// TIA Portal V18 export
// export: Created 2025-12-01T17:50:27.3546256Z, ExportSetting None, DisplayName Totally Integrated Automation Portal, DisplayVersion V18 Update 5, DisplayName TIA Portal Openness, DisplayVersion V18 Update 5, DisplayName TIA Portal Teamcenter Gateway, DisplayVersion V18, DisplayName TIA Portal Version Control Interface, DisplayVersion V18, DisplayName STEP 7 Professional, DisplayVersion V18 Update 5, DisplayName STEP 7 Safety, DisplayVersion V18, DisplayName WinCC Professional, DisplayVersion V18 Update 5
FUNCTION "CheckData" : Void   // FC4023, SCL
{ S7_Optimized_Access := 'FALSE' }
// stored: AutoNumber false, SetENOAutomatically false
   VAR_INPUT
      DBNo : Int;
      DBBNO : Int;
      ByteLenth : Int;
   END_VAR
   VAR_OUTPUT
      AlarmON : Bool;
   END_VAR
   VAR_TEMP
      AlarmByte : Int;
      tByte : Int;
   END_VAR
BEGIN
   #AlarmON := 0;
   #AlarmByte := 0;
   IF #ByteLenth>0 THEN
       FOR #tByte:=0 TO #ByteLenth-1 DO
           IF PEEK_BYTE(area:=16#84,dbNumber:=#DBNo,byteOffset:=#DBBNO+#tByte)<>0 THEN
               #AlarmON := TRUE;
               #AlarmByte := #DBBNO + #tByte;
               EXIT;
           ELSE
               #AlarmON := false;
               #AlarmByte := 0;
           END_IF;
       END_FOR;
   END_IF;
END_FUNCTION
